(*

short summary
=============
A specialized candy. It can be consumed by any candy consumer.
It supports dynamic creation. Furthermore, it calls the method 
AbstractCandy.initializeDispatchers after FB_init.

legal notes
===========
SPDX-FileCopyrightText: © 2024 ekvip automation GmbH <info@ekvip.de>
SPDX-License-Identifier: Apache-2.0
For details check: Apache-2.0_

.. _Apache-2.0: https://www.apache.org/licenses/LICENSE-2.0

*)

{attribute 'enable_dynamic_creation'}
{attribute 'call_after_init'}
FUNCTION_BLOCK FINAL BrachsCandyCorn EXTENDS AbstractCandy
VAR_INPUT
END_VAR
VAR_OUTPUT
END_VAR
VAR
END_VAR

(*

short summary
=============
it initializes the amount, the candy name and 
the binary coded candy type  

legal notes
===========
SPDX-FileCopyrightText: © 2024 ekvip automation GmbH <info@ekvip.de>
SPDX-License-Identifier: Apache-2.0
For details check: Apache-2.0_

.. _Apache-2.0: https://www.apache.org/licenses/LICENSE-2.0

*)

METHOD FB_init :BOOL
VAR_INPUT
	(* if TRUE, the retain variables are initialized (warm start / cold start) *)
	bInitRetains	:BOOL;
	(* if TRUE, the instance afterwards gets moved into the copy code (online change) *)
	bInCopyCode		:BOOL;
END_VAR
THIS^.amount := 312;
THIS^.name := 'Brach$'s Candy Corn';
THIS^.candyType := CandyTypes.GUMMY_CANDY OR CandyTypes.CANDY_CORN;
END_METHOD

END_FUNCTION_BLOCK

(* stored: Version 1.1.0.1
   POU BrachsCandyCorn: Id {acd0bfca-ec4c-4c64-8b57-c4aaa41a0807}, SpecialFunc None
   Method FB_init: Id {6f83cd01-c435-48e0-910a-adc9ca030e13} *)
